FUNCTION_BLOCK FB_RPC
VAR_INPUT
END_VAR
VAR_OUTPUT
END_VAR
VAR
	callCntAddition : UINT;
	callCntReadString : UINT;
	callCntWriteString : UINT;
	callCntReadStruct : UINT;
	callCntWriteStruct : UINT;
	
	m_myType : T_MyType;
	
	fbMsg : FB_TcMessage;
END_VAR

{attribute 'TcRpcEnable':='1'}
METHOD Addition : UINT
VAR_INPUT
	val_a : UINT;
	val_b : UINT;
END_VAR
callCntAddition := callCntAddition + 1;
Addition := val_a + val_b;
END_METHOD

METHOD FB_init : BOOL
VAR_INPUT
	bInitRetains : BOOL; // if TRUE, the retain variables are initialized (warm start / cold start)
	bInCopyCode : BOOL;  // if TRUE, the instance afterwards gets moved into the copy code (online change)
END_VAR
fbMsg.CreateEx(TC_EVENTS.RpcEventClass.WriteString, 0);
END_METHOD

{attribute 'TcRpcEnable':='1'}
METHOD ReadString : STRING
VAR_INPUT
END_VAR
VAR
	s_string : STRING := 'ReadString: Current call count: ';
END_VAR
callCntReadString := callCntReadString +1;
ReadString := CONCAT(s_string, UDINT_TO_STRING(callCntReadString));
END_METHOD

{attribute 'TcRpcEnable':='1'}
METHOD ReadStruct : T_MyType
VAR_INPUT
END_VAR
callCntReadStruct := callCntReadStruct + 1;
ReadStruct := m_myType;
END_METHOD

{attribute 'TcRpcEnable':='1'}
METHOD WriteString
VAR_INPUT
	in : STRING;
END_VAR
callCntWriteString := callCntWriteString +1;
fbMsg.Send(0); 
//ADSLOGSTR(
//	msgCtrlMask := ADSLOG_MSGTYPE_WARN OR ADSLOG_MSGTYPE_LOG,
//	msgFmtStr := 'String received: %s',
//	strArg := in
//	);
END_METHOD

{attribute 'TcRpcEnable':='1'}
METHOD WriteStruct : UINT
VAR_INPUT
	in : T_MyType;
END_VAR
m_myType.a := in.a;
m_myType.b := in.b;
m_myType.c := in.c;
callCntWriteStruct := callCntWriteStruct + 1;
WriteStruct := callCntWriteStruct;
END_METHOD

END_FUNCTION_BLOCK

(* stored: Version 1.1.0.1, ProductVersion 3.1.4024.12
   POU FB_RPC: Id {802561c0-ad01-4453-87af-ef5a372c7100}, SpecialFunc None
   Method Addition: Id {219d4a37-3601-46c1-90e8-1dad808a66ee}
   Method FB_init: Id {c5c4e316-c12b-4ba3-b329-1e3bdffc3cd9}
   Method ReadString: Id {b09955d0-ae50-4305-b477-83977ac2d6e6}
   Method ReadStruct: Id {9b7d9754-9fa1-4a6a-8e13-bb5d1dc7ffb0}
   Method WriteString: Id {458a276f-107a-4255-bfdb-a52b030572e5}
   Method WriteStruct: Id {510d9dfd-6ff4-43a2-a074-eb1bea49f8b0} *)
